Universal Robots URScript: painter_robot.urscript

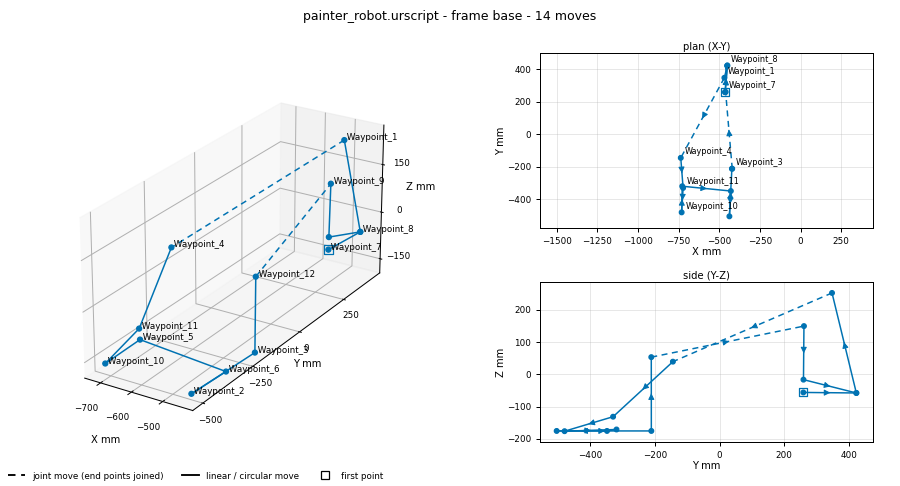
[picture p0: tool path of painter_robot.urscript in frame base, 14 of 15 moves have a stored position in this frame; points joined in program order, loops and branches not executed]
global Waypoint_9_p=p[-.461153166603, .261404301903, .149701904930, -1.147428535791, 1.265411452576, 1.154438243047]
global Waypoint_9_q=[3.492734432220459, -1.8469163380064906, -2.3516767024993896, -2.0640469990172328, 0.43328016996383667, -1.573874298726217]
global Waypoint_7_p=p[-.464409338493, .259576740704, -.055872861389, -1.147437155644, 1.265495473765, 1.154537514520]
global Waypoint_7_q=[3.493987560272217, -2.3023678265013636, -2.3362555503845215, -1.6231171093382777, 0.4341811239719391, -1.574737850819723]
global Waypoint_8_p=p[-.450748021250, .423734398792, -.057515019471, -1.147448426614, 1.265406205188, 1.154461724981]
global Waypoint_8_q=[3.1480305194854736, -2.308702131310934, -2.3212225437164307, -1.5532189563712855, 0.08862350881099701, -1.6554549376117151]
global Waypoint_1_p=p[-.468754199091, .348377937837, .252407934264, -1.205918416475, 1.206115090294, 1.188293286133]
global Waypoint_1_q=[3.313075065612793, -1.6692053280272425, -2.2915329933166504, -2.329076429406637, 0.18499808013439178, -1.5778215567218226]
global Waypoint_4_p=p[-.737242567318, -.144664408931, .039487065289, 1.171044697935, -1.230260213529, 1.160856073330]
global Waypoint_4_q=[3.230626106262207, -2.291882177392477, -1.850191354751587, -2.1618010006346644, -2.9962649981128138, 1.5419538021087646]
global Waypoint_11_p=p[-.722929201211, -.329900380655, -.131047981180, 1.171110635473, -1.230129715872, 1.160842456842]
global Waypoint_11_q=[3.493828773498535, -2.5374542675414027, -1.839306354522705, -1.9127589664854945, -2.733563486729757, 1.5559415817260742]
global Waypoint_10_p=p[-.731901180419, -.480277059314, -.175951285082, 1.171099620279, -1.230187489129, 1.160865956328]
global Waypoint_10_q=[3.6793060302734375, -2.6311007938780726, -1.726177453994751, -1.930340429345602, -2.5482190291034144, 1.5576369762420654]
global Waypoint_5_p=p[-.728138968366, -.319357666912, -.170624304961, 1.160803801776, -1.244838978120, 1.176020382525]
global Waypoint_5_q=[3.47694730758667, -2.6031304798521937, -1.8057928085327148, -1.8808347187437953, -2.750449244176046, 1.5763094425201416]
global Waypoint_6_p=p[-.428989668466, -.348779387942, -.175148595083, 1.171394707874, -1.229332244707, 1.160108321183]
global Waypoint_6_q=[3.787374496459961, -2.5929767094054164, -2.3563084602355957, -1.3351410192302247, -2.439634148274557, 1.5601999759674072]
global Waypoint_2_p=p[-.437902153645, -.504759143613, -.175178763808, 1.171371798126, -1.229497272785, 1.160177992084]
global Waypoint_2_q=[4.036845684051514, -2.566859861413473, -2.2385849952697754, -1.4788636428168793, -2.1902945677386683, 1.5602145195007324]
global Waypoint_3_p=p[-.422545960905, -.211443417247, -.175149994135, 1.171380838322, -1.229394092031, 1.160088186029]
global Waypoint_3_q=[3.47505521774292, -2.602645059625143, -2.381822347640991, -1.3011088234237214, -2.751882616673605, 1.5592272281646729]
global Waypoint_12_p=p[-.420457502621, -.211594888413, .053507108638, 1.171396003079, -1.229477743479, 1.160244204073]
global Waypoint_12_q=[3.477740526199341, -2.0118681393065394, -2.5099258422851562, -1.7644521198668421, -2.7490766684161585, 1.5586540699005127]
global Waypoint_13_p=p[-.463734707648, .259947276897, -.016236930022, -1.147428673602, 1.265426779328, 1.154480799509]
global Waypoint_13_q=[3.493776321411133, -2.212206026116842, -2.3524715900421143, -1.6972547970213832, 0.43404772877693176, -1.5746172110186976]



def pickAndPlace():
    # twofg_release(width=71.00000000000001, speed=100, external_release=True, tool_index=0 )
    # twofg_payload_set(mass = 0.0, tool_index = 0, use_guard = False)
    # movel(Waypoint_9_p, t=0.5)
    movej(Waypoint_9_q, t= 0.7)
    movel(Waypoint_7_p, t=0.5)
    movel(Waypoint_8_p, a=1.2, v=0.15)
    # twofg_grip(width=45.400000000000006, force=50, speed=100, external_grip=True, stop_if_no_force=False, tool_index=0)
    # twofg_payload_set(mass = 0.0, tool_index = 0, use_guard = True)
    movel(Waypoint_1_p, t=0.6, r=0.05)
    movej(get_inverse_kin(Waypoint_4_p, qnear=Waypoint_4_q), t=0.9)
    movel(Waypoint_11_p, t=0.6)
    movel(Waypoint_10_p, a=1.2, v=0.25)
    # twofg_release(width=71.00000000000001, speed=100, external_release=True, tool_index=0 )
    # twofg_payload_set(mass = 0.0, tool_index = 0, use_guard = False)
    movel(Waypoint_5_p, a=1.2, v=0.15)
    movel(Waypoint_6_p, t=0.4)
    movel(Waypoint_2_p, a=1.2, v=0.15)
    # twofg_grip(width=46.0, force=50, speed=100, external_grip=True, stop_if_no_force=False, tool_index=0)
    # twofg_payload_set(mass = 0.0, tool_index = 0, use_guard = False)
    movel(Waypoint_3_p, t=0.5)
    movel(Waypoint_12_p, t=0.6)
    movej(get_inverse_kin(Waypoint_9_p, qnear=Waypoint_9_q), t=0.8)
    movel(Waypoint_13_p, t=0.6)
    movel(Waypoint_8_p, t=1.5)
    # twofg_release(width=71.00000000000001, speed=100, external_release=True, tool_index=0 )
    # twofg_payload_set(mass = 0.0, tool_index = 0, use_guard = False)
end

pickAndPlace()
